(* Logix 5000 project; controller BTS01 vendor 1 type 14 code 217 rev 32.14; software revision 32.04; part 4 of 15 *)
(* tags used below, declared in another part *)
   Alarm_Active : DINT;
   Alarm_TMR : TIMER[17,32];
   ALM_ENABLE : DINT[25];
   HMI_Global_Alarm_Ack_PB : BOOL;
   HMIAlarms : DINT[25];   // Alarm Trigger Array
   HMIAlarmsMsg : STRING64[17,32];   // Alarm Descriptions to Match Alarm Trigger Array
(* Alarm, continued *)

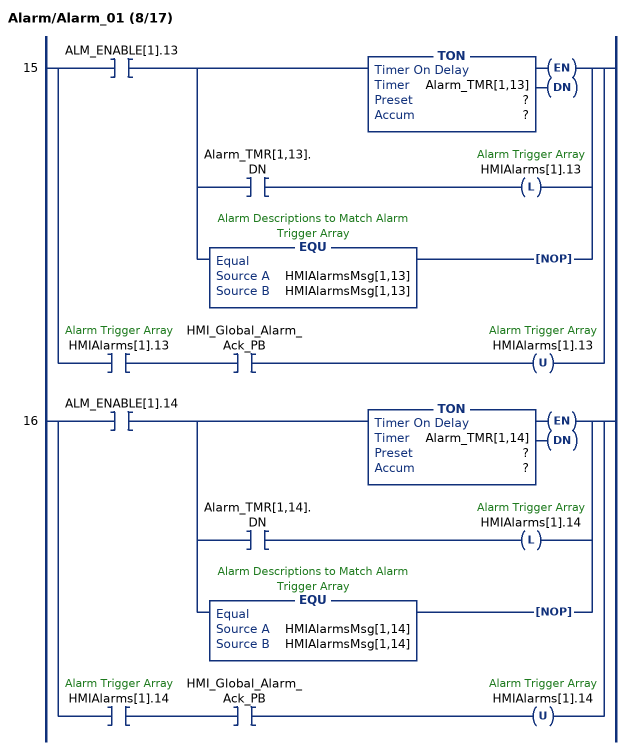
   [picture p45: Alarm/Alarm_01 rungs 15-16]
   15: [XIC(ALM_ENABLE[1].13) [TON(Alarm_TMR[1,13],?,?) ,XIC(Alarm_TMR[1,13].DN) OTL(HMIAlarms[1].13) ,EQU(HMIAlarmsMsg[1,13],HMIAlarmsMsg[1,13]) NOP() ] ,XIC(HMIAlarms[1].13) XIC(HMI_Global_Alarm_Ack_PB) OTU(HMIAlarms[1].13) ];
   16: [XIC(ALM_ENABLE[1].14) [TON(Alarm_TMR[1,14],?,?) ,XIC(Alarm_TMR[1,14].DN) OTL(HMIAlarms[1].14) ,EQU(HMIAlarmsMsg[1,14],HMIAlarmsMsg[1,14]) NOP() ] ,XIC(HMIAlarms[1].14) XIC(HMI_Global_Alarm_Ack_PB) OTU(HMIAlarms[1].14) ];
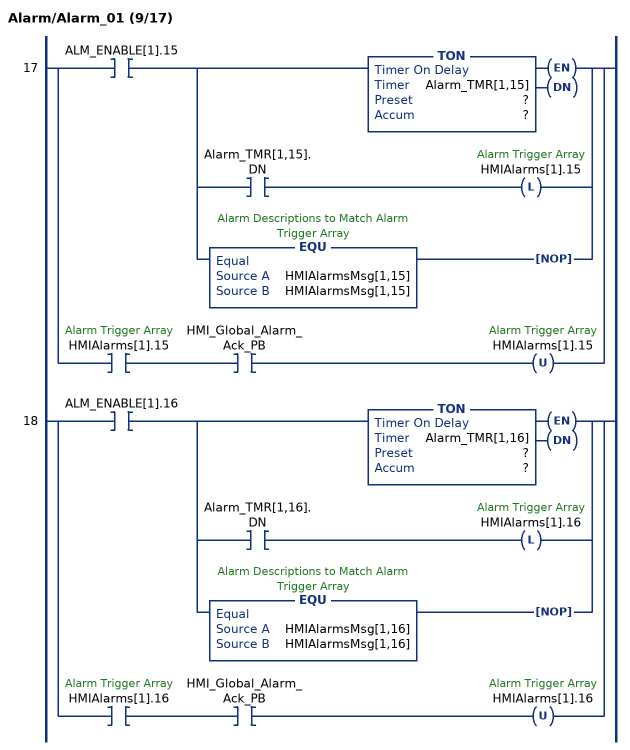
   17: [XIC(ALM_ENABLE[1].15) [TON(Alarm_TMR[1,15],?,?) ,XIC(Alarm_TMR[1,15].DN) OTL(HMIAlarms[1].15) ,EQU(HMIAlarmsMsg[1,15],HMIAlarmsMsg[1,15]) NOP() ] ,XIC(HMIAlarms[1].15) XIC(HMI_Global_Alarm_Ack_PB) OTU(HMIAlarms[1].15) ];
   18: [XIC(ALM_ENABLE[1].16) [TON(Alarm_TMR[1,16],?,?) ,XIC(Alarm_TMR[1,16].DN) OTL(HMIAlarms[1].16) ,EQU(HMIAlarmsMsg[1,16],HMIAlarmsMsg[1,16]) NOP() ] ,XIC(HMIAlarms[1].16) XIC(HMI_Global_Alarm_Ack_PB) OTU(HMIAlarms[1].16) ];
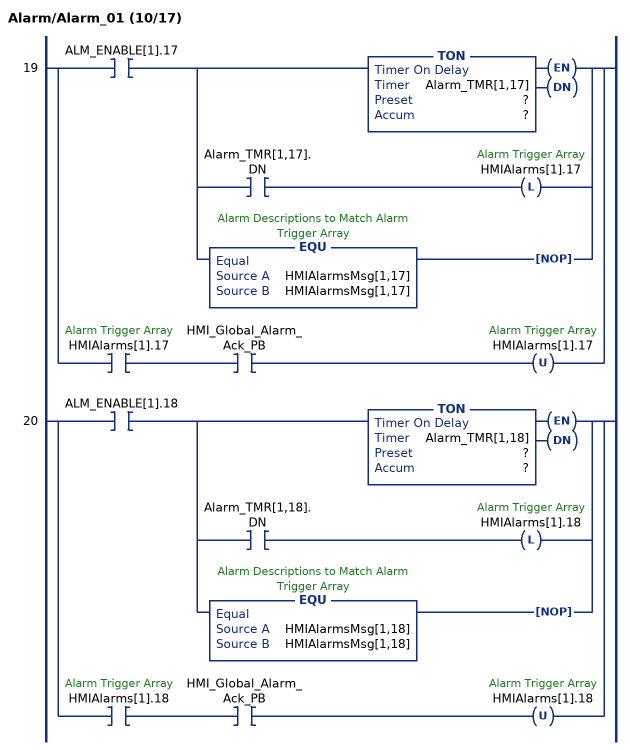
   19: [XIC(ALM_ENABLE[1].17) [TON(Alarm_TMR[1,17],?,?) ,XIC(Alarm_TMR[1,17].DN) OTL(HMIAlarms[1].17) ,EQU(HMIAlarmsMsg[1,17],HMIAlarmsMsg[1,17]) NOP() ] ,XIC(HMIAlarms[1].17) XIC(HMI_Global_Alarm_Ack_PB) OTU(HMIAlarms[1].17) ];
   20: [XIC(ALM_ENABLE[1].18) [TON(Alarm_TMR[1,18],?,?) ,XIC(Alarm_TMR[1,18].DN) OTL(HMIAlarms[1].18) ,EQU(HMIAlarmsMsg[1,18],HMIAlarmsMsg[1,18]) NOP() ] ,XIC(HMIAlarms[1].18) XIC(HMI_Global_Alarm_Ack_PB) OTU(HMIAlarms[1].18) ];
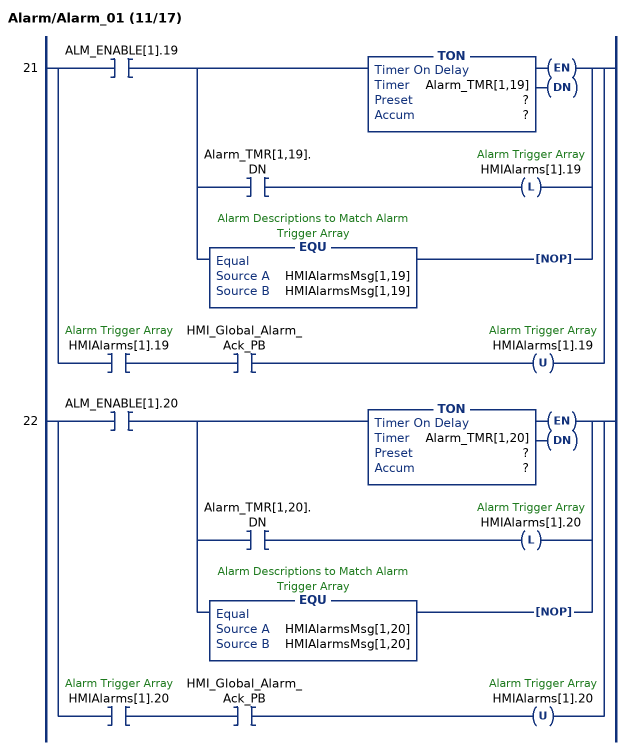
   21: [XIC(ALM_ENABLE[1].19) [TON(Alarm_TMR[1,19],?,?) ,XIC(Alarm_TMR[1,19].DN) OTL(HMIAlarms[1].19) ,EQU(HMIAlarmsMsg[1,19],HMIAlarmsMsg[1,19]) NOP() ] ,XIC(HMIAlarms[1].19) XIC(HMI_Global_Alarm_Ack_PB) OTU(HMIAlarms[1].19) ];
   22: [XIC(ALM_ENABLE[1].20) [TON(Alarm_TMR[1,20],?,?) ,XIC(Alarm_TMR[1,20].DN) OTL(HMIAlarms[1].20) ,EQU(HMIAlarmsMsg[1,20],HMIAlarmsMsg[1,20]) NOP() ] ,XIC(HMIAlarms[1].20) XIC(HMI_Global_Alarm_Ack_PB) OTU(HMIAlarms[1].20) ];
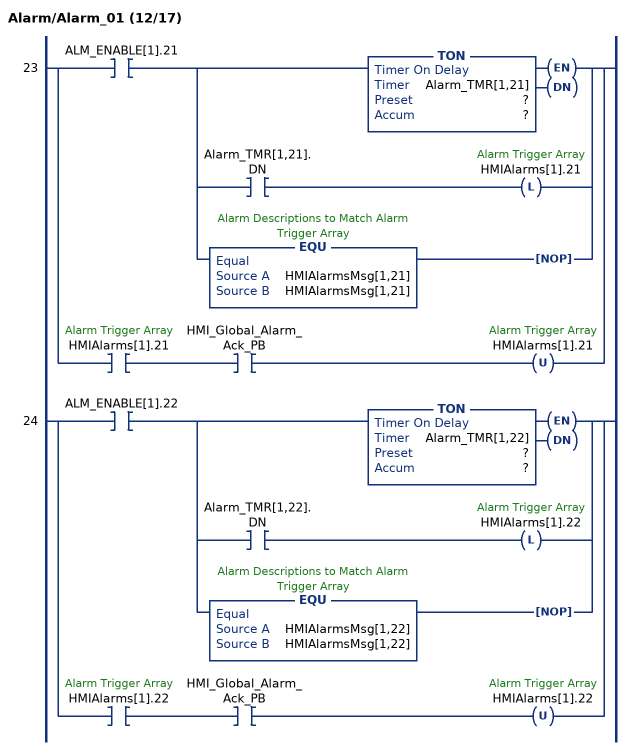
   23: [XIC(ALM_ENABLE[1].21) [TON(Alarm_TMR[1,21],?,?) ,XIC(Alarm_TMR[1,21].DN) OTL(HMIAlarms[1].21) ,EQU(HMIAlarmsMsg[1,21],HMIAlarmsMsg[1,21]) NOP() ] ,XIC(HMIAlarms[1].21) XIC(HMI_Global_Alarm_Ack_PB) OTU(HMIAlarms[1].21) ];
   24: [XIC(ALM_ENABLE[1].22) [TON(Alarm_TMR[1,22],?,?) ,XIC(Alarm_TMR[1,22].DN) OTL(HMIAlarms[1].22) ,EQU(HMIAlarmsMsg[1,22],HMIAlarmsMsg[1,22]) NOP() ] ,XIC(HMIAlarms[1].22) XIC(HMI_Global_Alarm_Ack_PB) OTU(HMIAlarms[1].22) ];
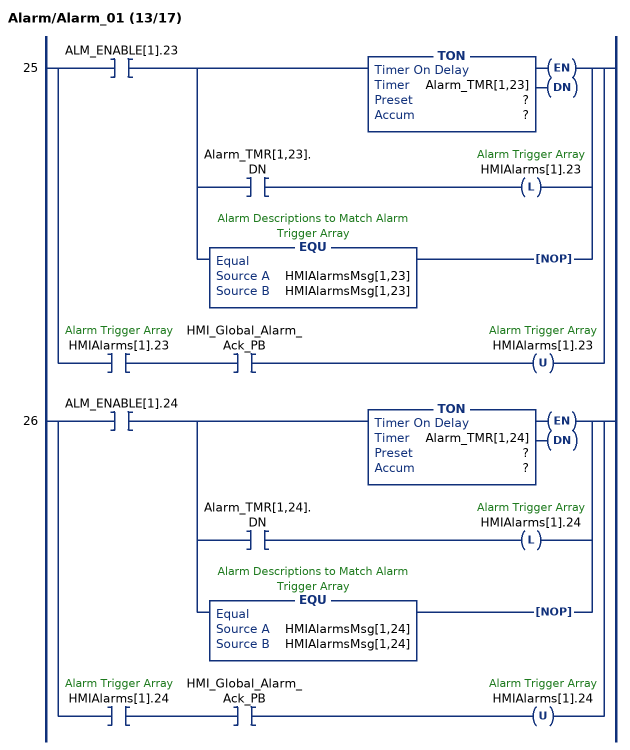
   25: [XIC(ALM_ENABLE[1].23) [TON(Alarm_TMR[1,23],?,?) ,XIC(Alarm_TMR[1,23].DN) OTL(HMIAlarms[1].23) ,EQU(HMIAlarmsMsg[1,23],HMIAlarmsMsg[1,23]) NOP() ] ,XIC(HMIAlarms[1].23) XIC(HMI_Global_Alarm_Ack_PB) OTU(HMIAlarms[1].23) ];
   26: [XIC(ALM_ENABLE[1].24) [TON(Alarm_TMR[1,24],?,?) ,XIC(Alarm_TMR[1,24].DN) OTL(HMIAlarms[1].24) ,EQU(HMIAlarmsMsg[1,24],HMIAlarmsMsg[1,24]) NOP() ] ,XIC(HMIAlarms[1].24) XIC(HMI_Global_Alarm_Ack_PB) OTU(HMIAlarms[1].24) ];
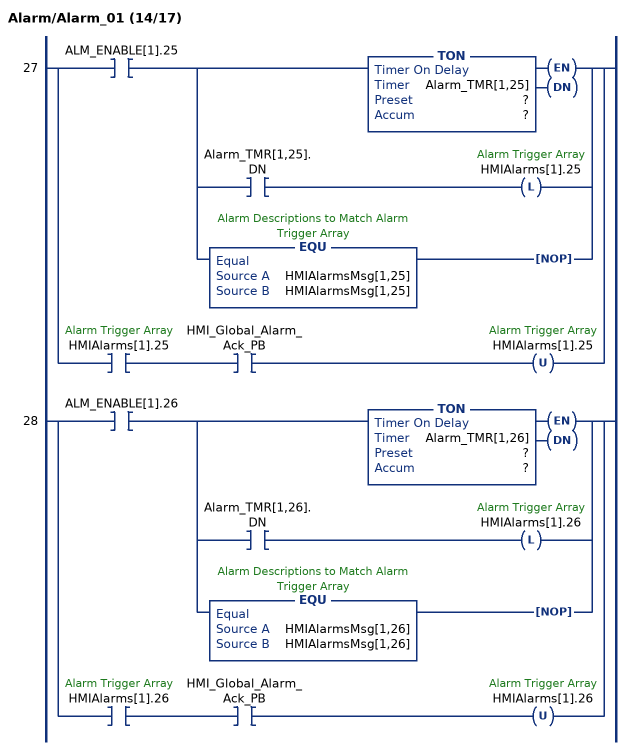
   27: [XIC(ALM_ENABLE[1].25) [TON(Alarm_TMR[1,25],?,?) ,XIC(Alarm_TMR[1,25].DN) OTL(HMIAlarms[1].25) ,EQU(HMIAlarmsMsg[1,25],HMIAlarmsMsg[1,25]) NOP() ] ,XIC(HMIAlarms[1].25) XIC(HMI_Global_Alarm_Ack_PB) OTU(HMIAlarms[1].25) ];
   28: [XIC(ALM_ENABLE[1].26) [TON(Alarm_TMR[1,26],?,?) ,XIC(Alarm_TMR[1,26].DN) OTL(HMIAlarms[1].26) ,EQU(HMIAlarmsMsg[1,26],HMIAlarmsMsg[1,26]) NOP() ] ,XIC(HMIAlarms[1].26) XIC(HMI_Global_Alarm_Ack_PB) OTU(HMIAlarms[1].26) ];
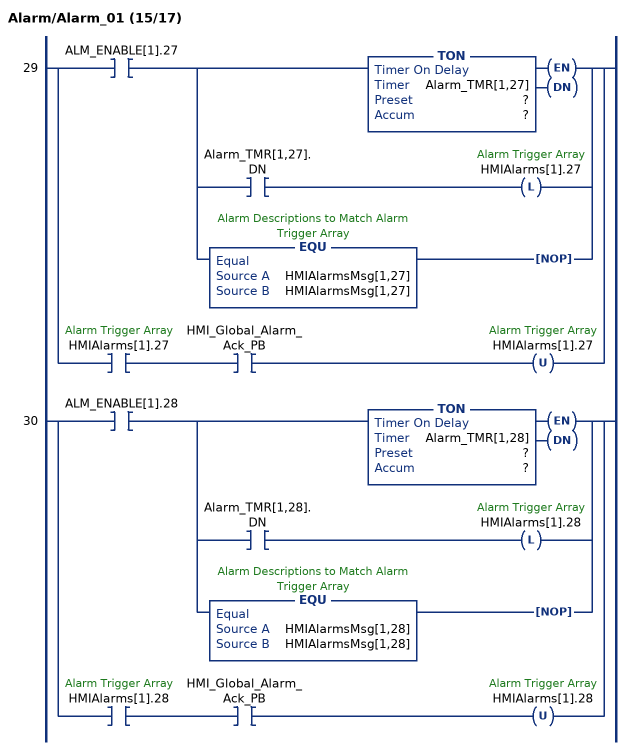
   29: [XIC(ALM_ENABLE[1].27) [TON(Alarm_TMR[1,27],?,?) ,XIC(Alarm_TMR[1,27].DN) OTL(HMIAlarms[1].27) ,EQU(HMIAlarmsMsg[1,27],HMIAlarmsMsg[1,27]) NOP() ] ,XIC(HMIAlarms[1].27) XIC(HMI_Global_Alarm_Ack_PB) OTU(HMIAlarms[1].27) ];
   30: [XIC(ALM_ENABLE[1].28) [TON(Alarm_TMR[1,28],?,?) ,XIC(Alarm_TMR[1,28].DN) OTL(HMIAlarms[1].28) ,EQU(HMIAlarmsMsg[1,28],HMIAlarmsMsg[1,28]) NOP() ] ,XIC(HMIAlarms[1].28) XIC(HMI_Global_Alarm_Ack_PB) OTU(HMIAlarms[1].28) ];
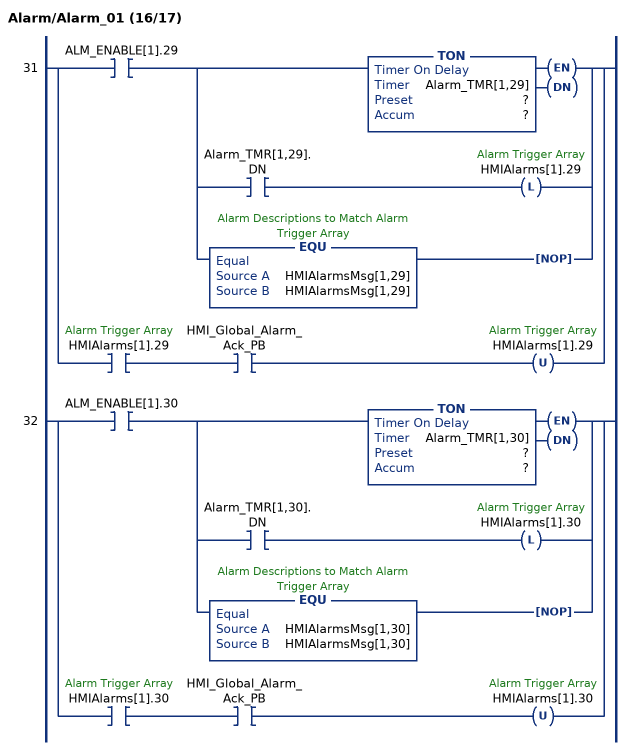
   31: [XIC(ALM_ENABLE[1].29) [TON(Alarm_TMR[1,29],?,?) ,XIC(Alarm_TMR[1,29].DN) OTL(HMIAlarms[1].29) ,EQU(HMIAlarmsMsg[1,29],HMIAlarmsMsg[1,29]) NOP() ] ,XIC(HMIAlarms[1].29) XIC(HMI_Global_Alarm_Ack_PB) OTU(HMIAlarms[1].29) ];
   32: [XIC(ALM_ENABLE[1].30) [TON(Alarm_TMR[1,30],?,?) ,XIC(Alarm_TMR[1,30].DN) OTL(HMIAlarms[1].30) ,EQU(HMIAlarmsMsg[1,30],HMIAlarmsMsg[1,30]) NOP() ] ,XIC(HMIAlarms[1].30) XIC(HMI_Global_Alarm_Ack_PB) OTU(HMIAlarms[1].30) ];
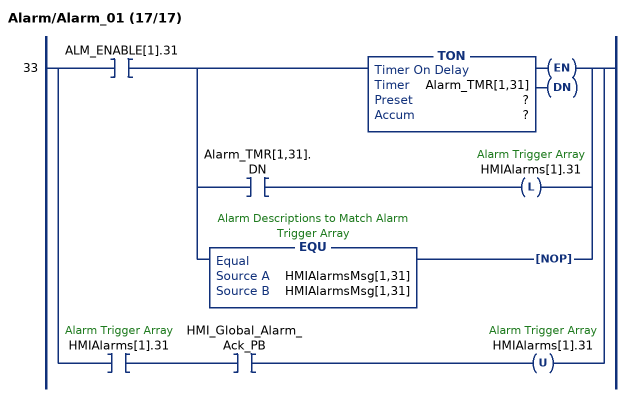
   33: [XIC(ALM_ENABLE[1].31) [TON(Alarm_TMR[1,31],?,?) ,XIC(Alarm_TMR[1,31].DN) OTL(HMIAlarms[1].31) ,EQU(HMIAlarmsMsg[1,31],HMIAlarmsMsg[1,31]) NOP() ] ,XIC(HMIAlarms[1].31) XIC(HMI_Global_Alarm_Ack_PB) OTU(HMIAlarms[1].31) ];
END_ROUTINE

ROUTINE Alarm_02   (* ladder *)
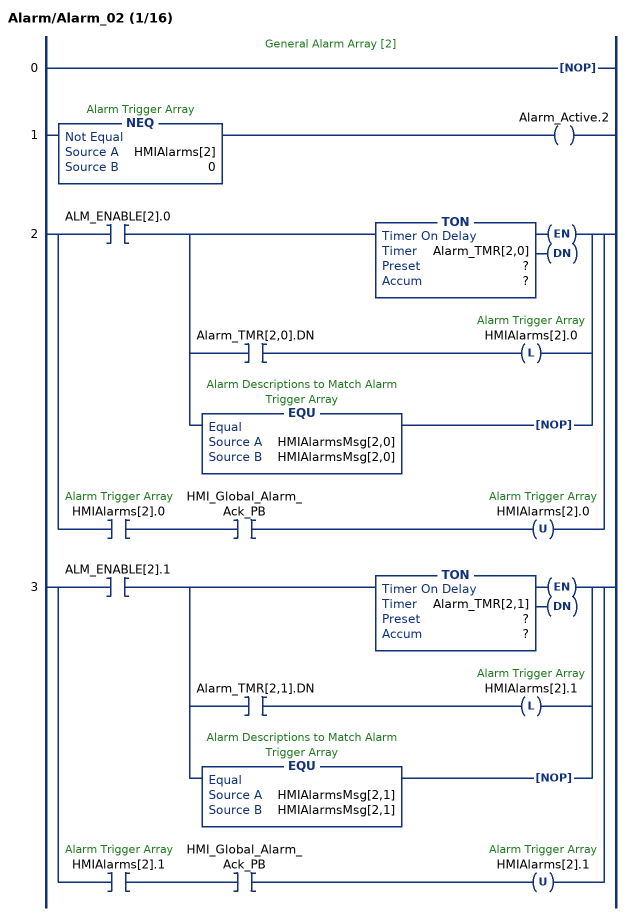
   // General Alarm Array [2]
   0: NOP();
   1: NEQ(HMIAlarms[2],0)OTE(Alarm_Active.2);
   2: [XIC(ALM_ENABLE[2].0) [TON(Alarm_TMR[2,0],?,?) ,XIC(Alarm_TMR[2,0].DN) OTL(HMIAlarms[2].0) ,EQU(HMIAlarmsMsg[2,0],HMIAlarmsMsg[2,0]) NOP() ] ,XIC(HMIAlarms[2].0) XIC(HMI_Global_Alarm_Ack_PB) OTU(HMIAlarms[2].0) ];
   3: [XIC(ALM_ENABLE[2].1) [TON(Alarm_TMR[2,1],?,?) ,XIC(Alarm_TMR[2,1].DN) OTL(HMIAlarms[2].1) ,EQU(HMIAlarmsMsg[2,1],HMIAlarmsMsg[2,1]) NOP() ] ,XIC(HMIAlarms[2].1) XIC(HMI_Global_Alarm_Ack_PB) OTU(HMIAlarms[2].1) ];
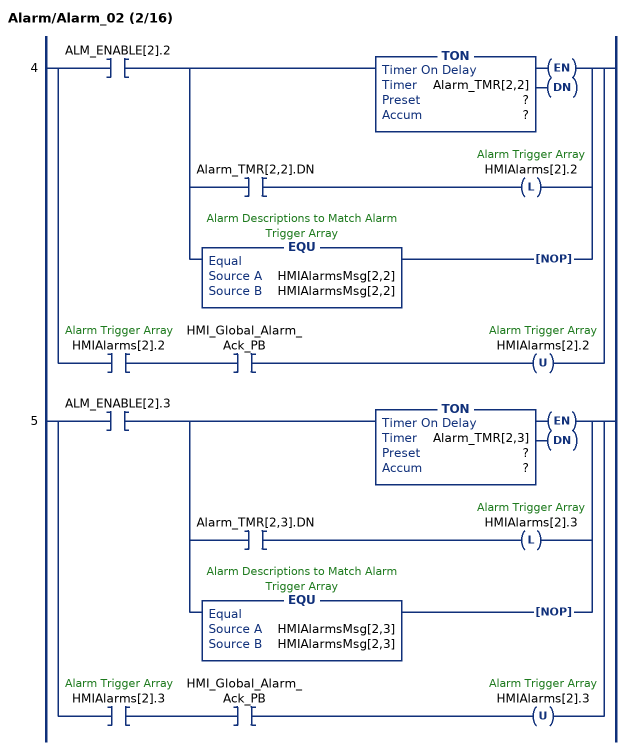
   4: [XIC(ALM_ENABLE[2].2) [TON(Alarm_TMR[2,2],?,?) ,XIC(Alarm_TMR[2,2].DN) OTL(HMIAlarms[2].2) ,EQU(HMIAlarmsMsg[2,2],HMIAlarmsMsg[2,2]) NOP() ] ,XIC(HMIAlarms[2].2) XIC(HMI_Global_Alarm_Ack_PB) OTU(HMIAlarms[2].2) ];
   5: [XIC(ALM_ENABLE[2].3) [TON(Alarm_TMR[2,3],?,?) ,XIC(Alarm_TMR[2,3].DN) OTL(HMIAlarms[2].3) ,EQU(HMIAlarmsMsg[2,3],HMIAlarmsMsg[2,3]) NOP() ] ,XIC(HMIAlarms[2].3) XIC(HMI_Global_Alarm_Ack_PB) OTU(HMIAlarms[2].3) ];
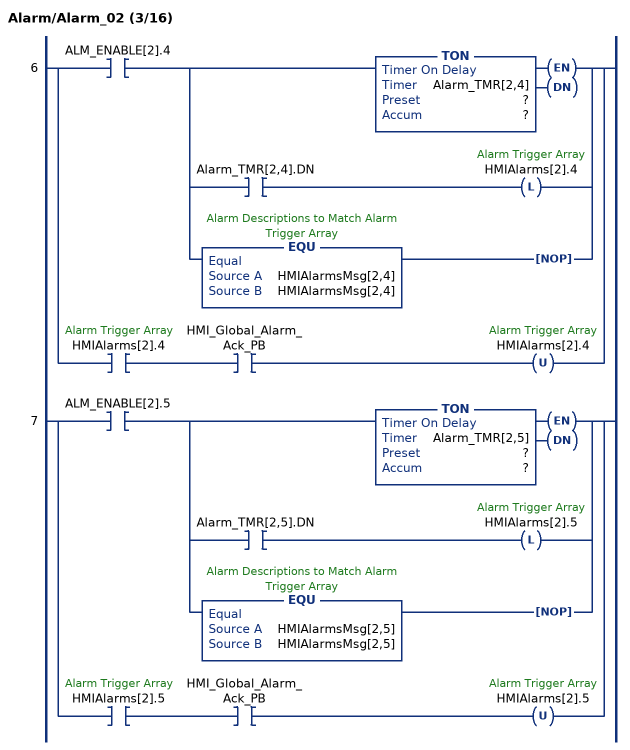
   6: [XIC(ALM_ENABLE[2].4) [TON(Alarm_TMR[2,4],?,?) ,XIC(Alarm_TMR[2,4].DN) OTL(HMIAlarms[2].4) ,EQU(HMIAlarmsMsg[2,4],HMIAlarmsMsg[2,4]) NOP() ] ,XIC(HMIAlarms[2].4) XIC(HMI_Global_Alarm_Ack_PB) OTU(HMIAlarms[2].4) ];
   7: [XIC(ALM_ENABLE[2].5) [TON(Alarm_TMR[2,5],?,?) ,XIC(Alarm_TMR[2,5].DN) OTL(HMIAlarms[2].5) ,EQU(HMIAlarmsMsg[2,5],HMIAlarmsMsg[2,5]) NOP() ] ,XIC(HMIAlarms[2].5) XIC(HMI_Global_Alarm_Ack_PB) OTU(HMIAlarms[2].5) ];
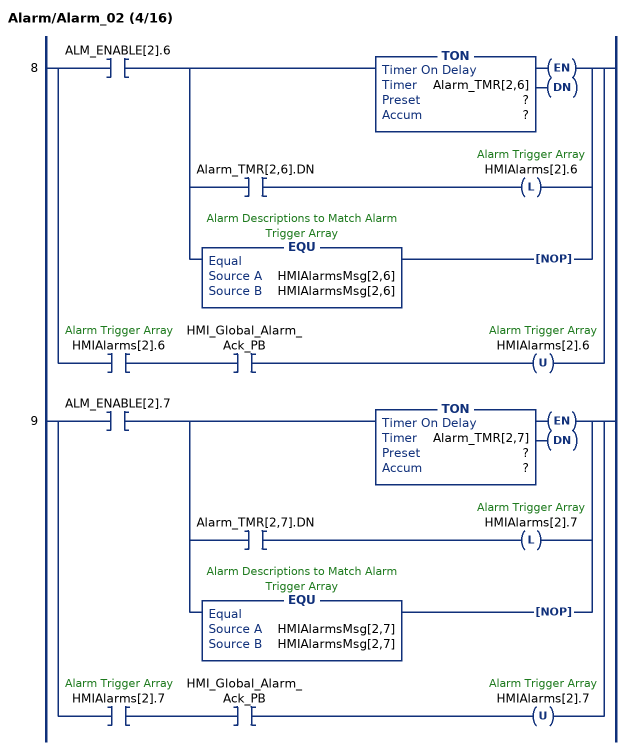
   8: [XIC(ALM_ENABLE[2].6) [TON(Alarm_TMR[2,6],?,?) ,XIC(Alarm_TMR[2,6].DN) OTL(HMIAlarms[2].6) ,EQU(HMIAlarmsMsg[2,6],HMIAlarmsMsg[2,6]) NOP() ] ,XIC(HMIAlarms[2].6) XIC(HMI_Global_Alarm_Ack_PB) OTU(HMIAlarms[2].6) ];
   9: [XIC(ALM_ENABLE[2].7) [TON(Alarm_TMR[2,7],?,?) ,XIC(Alarm_TMR[2,7].DN) OTL(HMIAlarms[2].7) ,EQU(HMIAlarmsMsg[2,7],HMIAlarmsMsg[2,7]) NOP() ] ,XIC(HMIAlarms[2].7) XIC(HMI_Global_Alarm_Ack_PB) OTU(HMIAlarms[2].7) ];
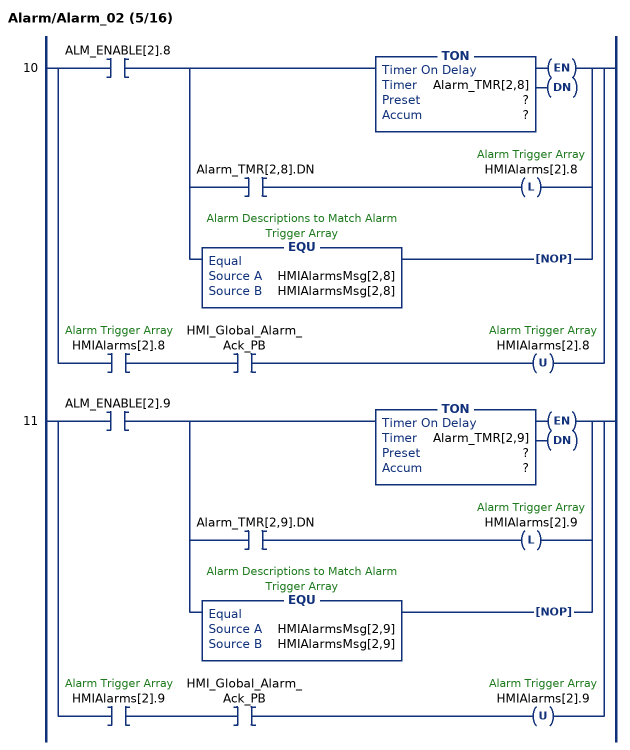
   10: [XIC(ALM_ENABLE[2].8) [TON(Alarm_TMR[2,8],?,?) ,XIC(Alarm_TMR[2,8].DN) OTL(HMIAlarms[2].8) ,EQU(HMIAlarmsMsg[2,8],HMIAlarmsMsg[2,8]) NOP() ] ,XIC(HMIAlarms[2].8) XIC(HMI_Global_Alarm_Ack_PB) OTU(HMIAlarms[2].8) ];
   11: [XIC(ALM_ENABLE[2].9) [TON(Alarm_TMR[2,9],?,?) ,XIC(Alarm_TMR[2,9].DN) OTL(HMIAlarms[2].9) ,EQU(HMIAlarmsMsg[2,9],HMIAlarmsMsg[2,9]) NOP() ] ,XIC(HMIAlarms[2].9) XIC(HMI_Global_Alarm_Ack_PB) OTU(HMIAlarms[2].9) ];
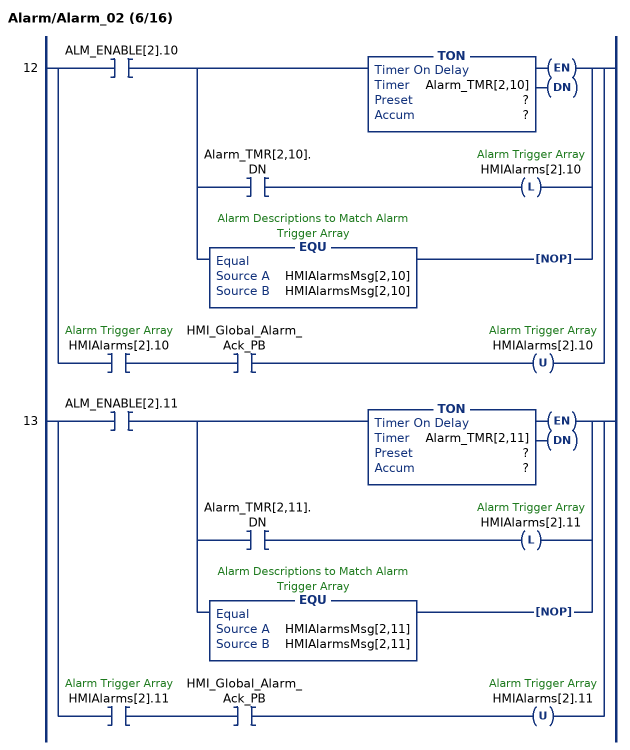
   12: [XIC(ALM_ENABLE[2].10) [TON(Alarm_TMR[2,10],?,?) ,XIC(Alarm_TMR[2,10].DN) OTL(HMIAlarms[2].10) ,EQU(HMIAlarmsMsg[2,10],HMIAlarmsMsg[2,10]) NOP() ] ,XIC(HMIAlarms[2].10) XIC(HMI_Global_Alarm_Ack_PB) OTU(HMIAlarms[2].10) ];
   13: [XIC(ALM_ENABLE[2].11) [TON(Alarm_TMR[2,11],?,?) ,XIC(Alarm_TMR[2,11].DN) OTL(HMIAlarms[2].11) ,EQU(HMIAlarmsMsg[2,11],HMIAlarmsMsg[2,11]) NOP() ] ,XIC(HMIAlarms[2].11) XIC(HMI_Global_Alarm_Ack_PB) OTU(HMIAlarms[2].11) ];
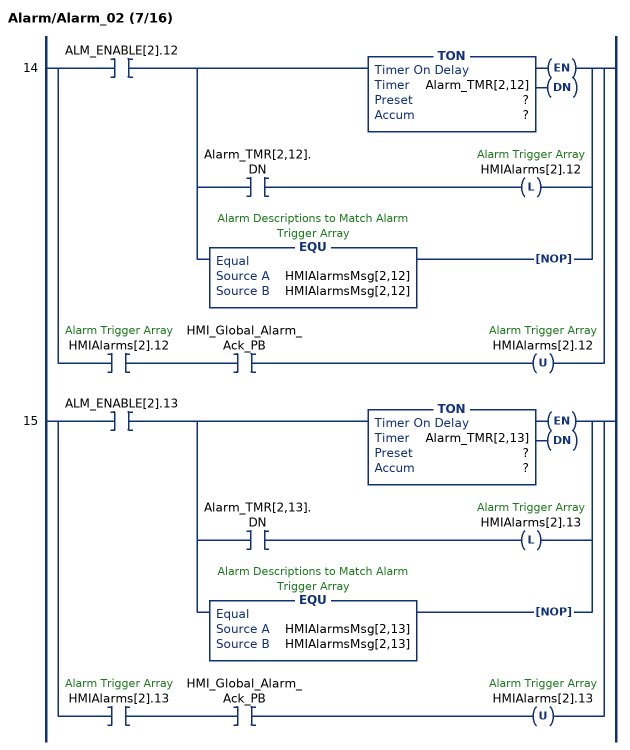
   14: [XIC(ALM_ENABLE[2].12) [TON(Alarm_TMR[2,12],?,?) ,XIC(Alarm_TMR[2,12].DN) OTL(HMIAlarms[2].12) ,EQU(HMIAlarmsMsg[2,12],HMIAlarmsMsg[2,12]) NOP() ] ,XIC(HMIAlarms[2].12) XIC(HMI_Global_Alarm_Ack_PB) OTU(HMIAlarms[2].12) ];
   15: [XIC(ALM_ENABLE[2].13) [TON(Alarm_TMR[2,13],?,?) ,XIC(Alarm_TMR[2,13].DN) OTL(HMIAlarms[2].13) ,EQU(HMIAlarmsMsg[2,13],HMIAlarmsMsg[2,13]) NOP() ] ,XIC(HMIAlarms[2].13) XIC(HMI_Global_Alarm_Ack_PB) OTU(HMIAlarms[2].13) ];
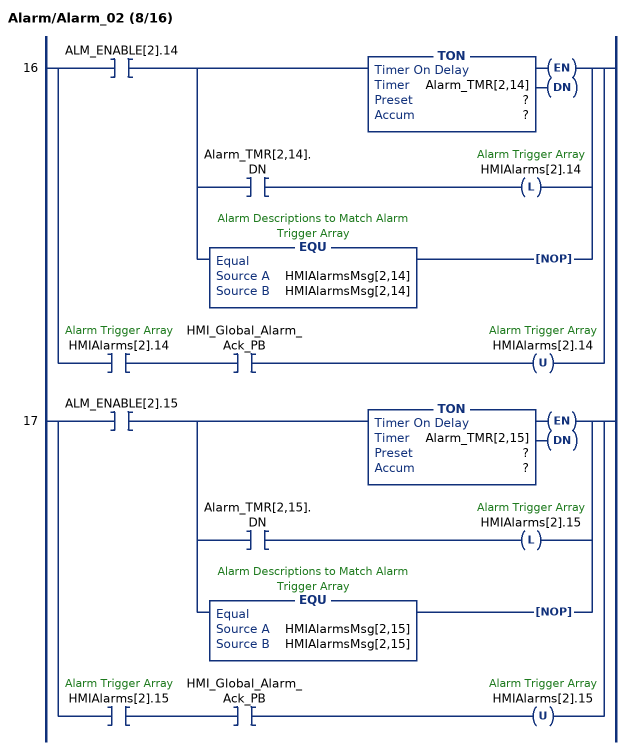
   16: [XIC(ALM_ENABLE[2].14) [TON(Alarm_TMR[2,14],?,?) ,XIC(Alarm_TMR[2,14].DN) OTL(HMIAlarms[2].14) ,EQU(HMIAlarmsMsg[2,14],HMIAlarmsMsg[2,14]) NOP() ] ,XIC(HMIAlarms[2].14) XIC(HMI_Global_Alarm_Ack_PB) OTU(HMIAlarms[2].14) ];
   17: [XIC(ALM_ENABLE[2].15) [TON(Alarm_TMR[2,15],?,?) ,XIC(Alarm_TMR[2,15].DN) OTL(HMIAlarms[2].15) ,EQU(HMIAlarmsMsg[2,15],HMIAlarmsMsg[2,15]) NOP() ] ,XIC(HMIAlarms[2].15) XIC(HMI_Global_Alarm_Ack_PB) OTU(HMIAlarms[2].15) ];
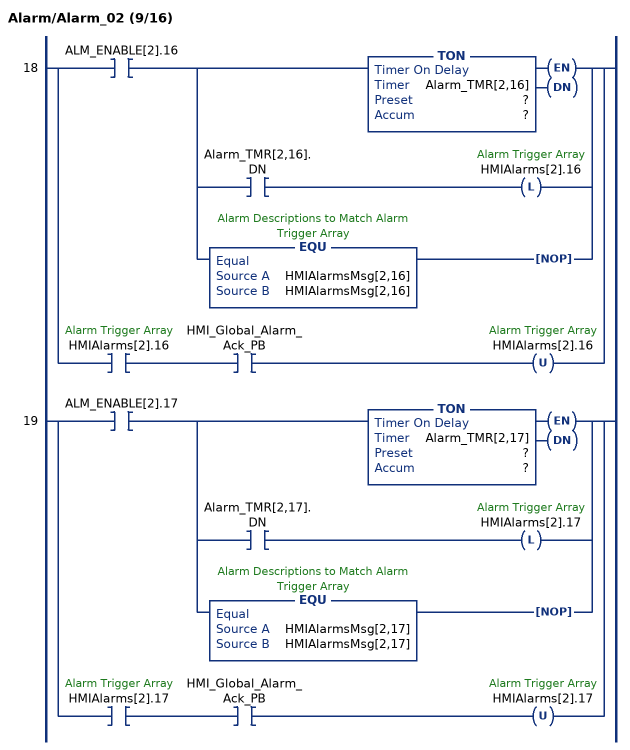
   18: [XIC(ALM_ENABLE[2].16) [TON(Alarm_TMR[2,16],?,?) ,XIC(Alarm_TMR[2,16].DN) OTL(HMIAlarms[2].16) ,EQU(HMIAlarmsMsg[2,16],HMIAlarmsMsg[2,16]) NOP() ] ,XIC(HMIAlarms[2].16) XIC(HMI_Global_Alarm_Ack_PB) OTU(HMIAlarms[2].16) ];
   19: [XIC(ALM_ENABLE[2].17) [TON(Alarm_TMR[2,17],?,?) ,XIC(Alarm_TMR[2,17].DN) OTL(HMIAlarms[2].17) ,EQU(HMIAlarmsMsg[2,17],HMIAlarmsMsg[2,17]) NOP() ] ,XIC(HMIAlarms[2].17) XIC(HMI_Global_Alarm_Ack_PB) OTU(HMIAlarms[2].17) ];
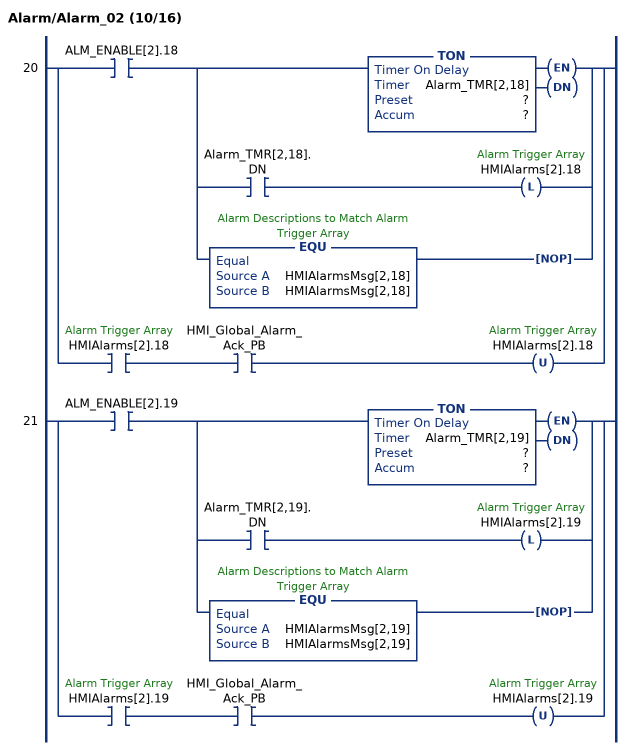
   20: [XIC(ALM_ENABLE[2].18) [TON(Alarm_TMR[2,18],?,?) ,XIC(Alarm_TMR[2,18].DN) OTL(HMIAlarms[2].18) ,EQU(HMIAlarmsMsg[2,18],HMIAlarmsMsg[2,18]) NOP() ] ,XIC(HMIAlarms[2].18) XIC(HMI_Global_Alarm_Ack_PB) OTU(HMIAlarms[2].18) ];
   21: [XIC(ALM_ENABLE[2].19) [TON(Alarm_TMR[2,19],?,?) ,XIC(Alarm_TMR[2,19].DN) OTL(HMIAlarms[2].19) ,EQU(HMIAlarmsMsg[2,19],HMIAlarmsMsg[2,19]) NOP() ] ,XIC(HMIAlarms[2].19) XIC(HMI_Global_Alarm_Ack_PB) OTU(HMIAlarms[2].19) ];
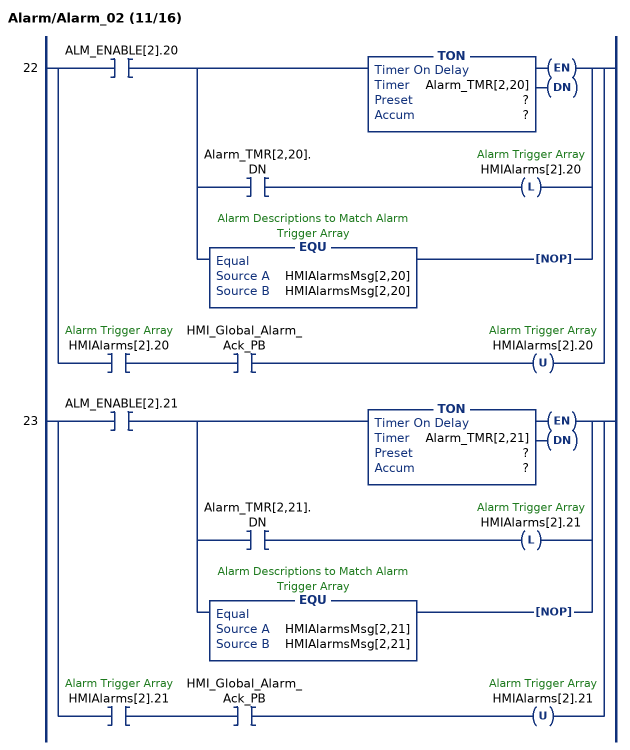
   22: [XIC(ALM_ENABLE[2].20) [TON(Alarm_TMR[2,20],?,?) ,XIC(Alarm_TMR[2,20].DN) OTL(HMIAlarms[2].20) ,EQU(HMIAlarmsMsg[2,20],HMIAlarmsMsg[2,20]) NOP() ] ,XIC(HMIAlarms[2].20) XIC(HMI_Global_Alarm_Ack_PB) OTU(HMIAlarms[2].20) ];
   23: [XIC(ALM_ENABLE[2].21) [TON(Alarm_TMR[2,21],?,?) ,XIC(Alarm_TMR[2,21].DN) OTL(HMIAlarms[2].21) ,EQU(HMIAlarmsMsg[2,21],HMIAlarmsMsg[2,21]) NOP() ] ,XIC(HMIAlarms[2].21) XIC(HMI_Global_Alarm_Ack_PB) OTU(HMIAlarms[2].21) ];
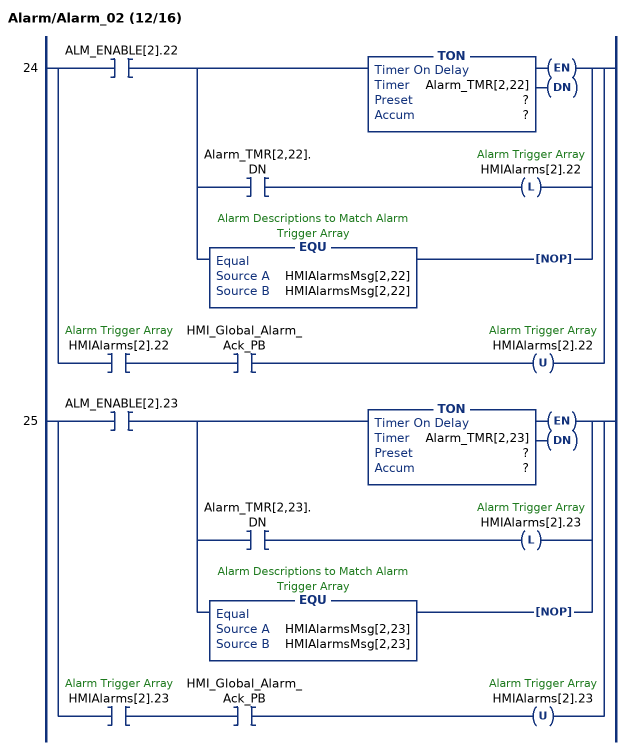
   24: [XIC(ALM_ENABLE[2].22) [TON(Alarm_TMR[2,22],?,?) ,XIC(Alarm_TMR[2,22].DN) OTL(HMIAlarms[2].22) ,EQU(HMIAlarmsMsg[2,22],HMIAlarmsMsg[2,22]) NOP() ] ,XIC(HMIAlarms[2].22) XIC(HMI_Global_Alarm_Ack_PB) OTU(HMIAlarms[2].22) ];
   25: [XIC(ALM_ENABLE[2].23) [TON(Alarm_TMR[2,23],?,?) ,XIC(Alarm_TMR[2,23].DN) OTL(HMIAlarms[2].23) ,EQU(HMIAlarmsMsg[2,23],HMIAlarmsMsg[2,23]) NOP() ] ,XIC(HMIAlarms[2].23) XIC(HMI_Global_Alarm_Ack_PB) OTU(HMIAlarms[2].23) ];
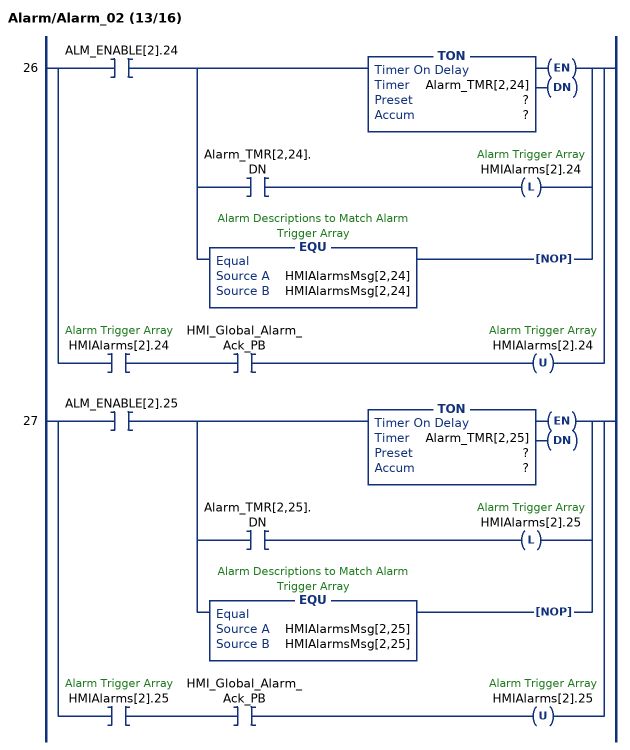
   26: [XIC(ALM_ENABLE[2].24) [TON(Alarm_TMR[2,24],?,?) ,XIC(Alarm_TMR[2,24].DN) OTL(HMIAlarms[2].24) ,EQU(HMIAlarmsMsg[2,24],HMIAlarmsMsg[2,24]) NOP() ] ,XIC(HMIAlarms[2].24) XIC(HMI_Global_Alarm_Ack_PB) OTU(HMIAlarms[2].24) ];
   27: [XIC(ALM_ENABLE[2].25) [TON(Alarm_TMR[2,25],?,?) ,XIC(Alarm_TMR[2,25].DN) OTL(HMIAlarms[2].25) ,EQU(HMIAlarmsMsg[2,25],HMIAlarmsMsg[2,25]) NOP() ] ,XIC(HMIAlarms[2].25) XIC(HMI_Global_Alarm_Ack_PB) OTU(HMIAlarms[2].25) ];
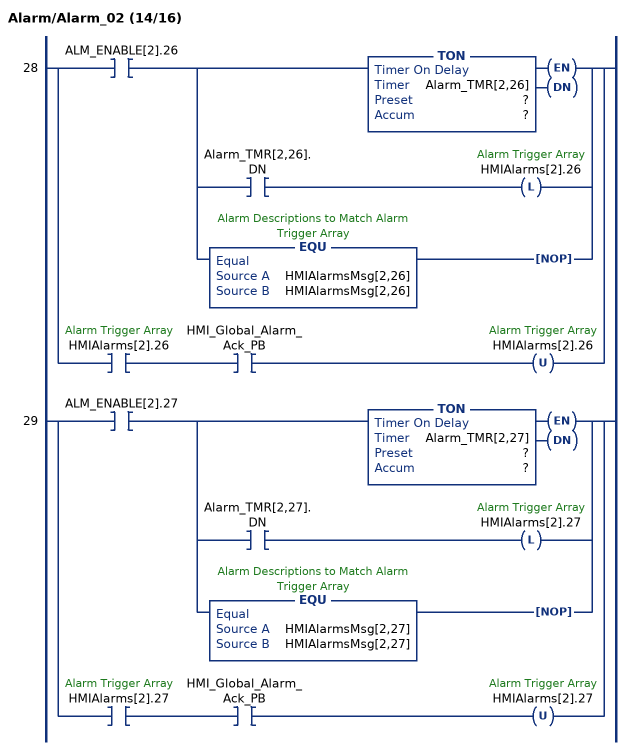
   28: [XIC(ALM_ENABLE[2].26) [TON(Alarm_TMR[2,26],?,?) ,XIC(Alarm_TMR[2,26].DN) OTL(HMIAlarms[2].26) ,EQU(HMIAlarmsMsg[2,26],HMIAlarmsMsg[2,26]) NOP() ] ,XIC(HMIAlarms[2].26) XIC(HMI_Global_Alarm_Ack_PB) OTU(HMIAlarms[2].26) ];
   29: [XIC(ALM_ENABLE[2].27) [TON(Alarm_TMR[2,27],?,?) ,XIC(Alarm_TMR[2,27].DN) OTL(HMIAlarms[2].27) ,EQU(HMIAlarmsMsg[2,27],HMIAlarmsMsg[2,27]) NOP() ] ,XIC(HMIAlarms[2].27) XIC(HMI_Global_Alarm_Ack_PB) OTU(HMIAlarms[2].27) ];
